FUNCTION_BLOCK FB_HomeReadSoftLimEnable
VAR_INPUT
	En: BOOL;
	bReset: BOOL;
    bExecute: BOOL;			
END_VAR
VAR_IN_OUT
	Axis: AXIS_REF;
END_VAR
VAR_OUTPUT
	EnO: BOOL;	
	bBusy: BOOL;
	bDone: BOOL;
	bError: BOOL;
	nErrorId: UDINT;	
	bSofLimEnableLow: BOOL:=TRUE;
	bSofLimEnableHigh: BOOL:=TRUE;
END_VAR
VAR
	fbReadSoftLimEnableLow:FB_ReadParameterInNc_v1_00;
	fbReadSoftLimEnableHigh:FB_ReadParameterInNc_v1_00;
END_VAR

En:=EnO;
IF bReset THEN
	bError:=FALSE;
	nErrorId:=0;
END_IF 
	
fbReadSoftLimEnableLow(
	bExecute:=bExecute,
	nDeviceGroup:= 16#5000,
	nIndexOffset:= 16#B,
	Axis:= Axis);

fbReadSoftLimEnableHigh(
	bExecute:=bExecute,
	nDeviceGroup:= 16#5000,
	nIndexOffset:= 16#C,
	Axis:= Axis);
	
bSofLimEnableLow:=DWORD_TO_BOOL(fbReadSoftLimEnableLow.nData);
bSofLimEnableHigh:=DWORD_TO_BOOL(fbReadSoftLimEnableHigh.nData);	

bBusy:=fbReadSoftLimEnableLow.bBusy OR fbReadSoftLimEnableHigh.bBusy;
bDone:=fbReadSoftLimEnableLow.bDone AND fbReadSoftLimEnableHigh.bDone AND bExecute;

bError:=fbReadSoftLimEnableLow.bError OR fbReadSoftLimEnableHigh.bError;
IF fbReadSoftLimEnableLow.bError THEN
  nErrorId:=fbReadSoftLimEnableLow.nErrorId;
ELSIF fbReadSoftLimEnableHigh.bError THEN
  nErrorId:=fbReadSoftLimEnableHigh.nErrorId;
END_IF

END_FUNCTION_BLOCK

(* stored: Version 1.1.0.1, ProductVersion 3.1.4022.10
   POU FB_HomeReadSoftLimEnable: Id {be900be5-0784-4633-94f1-38a4124c1620}, SpecialFunc None *)
